TYPE ST_SensirionFM :
STRUCT
	ctrl	:	ST_SensirionFMControl;
	stat	:	ST_SensirionFMStatus;
END_STRUCT
END_TYPE

(* stored: Version 1.1.0.1, ProductVersion 3.1.4018.5
   DUT ST_SensirionFM: Id {a6b8d86f-c2b0-4a79-92ac-31fbf668167c} *)
